FUNCTION_BLOCK FB_TestRound EXTENDS TcUnit.FB_TestSuite

testRoundReal();

METHOD testRoundReal
VAR
	rValue 		: REAL := 1000.555555;
	Actual		: REAL;
	Expected  	: REAL;
END_VAR
TEST('testRoundReal');

// Act
Actual := F_ROUNDREAL(rValue, 2); 

// Arrange
Expected := 1000.55;

// Assert
AssertEquals(Expected := Expected, 
			 Actual := Actual,
			 Message := 'testRoundReal Failed');
END_METHOD

END_FUNCTION_BLOCK

(* stored: Version 1.1.0.1, ProductVersion 3.1.4024.9
   POU FB_TestRound: Id {92000e0b-3a08-4346-91c0-8b471b1ff965}, SpecialFunc None
   Method testRoundReal: Id {972e2527-061b-4f8b-979d-4770a9b664a6} *)
